(* PLC project static_torsion.project, CODESYS CODESYS V3.5 SP17 Patch 3 *)
(* stored: creationDateTime 1970-01-01T00:00:00, modificationDateTime 2026-06-22T15:12:39.4699931 *)

PROGRAM MODBUS_DATA
  VAR
    MB_DI AT %MW40000 : WORD;  (* Входы дискретные модуль A11 (ECAT-2053) *)
    MB_TN AT %MW40001 : WORD;  (* Значение момента с АЦП модуля тензодатчика A14 (ECAT-2016N) *)
    MB_EN AT %MW40002 : ARRAY[0..1] OF WORD;  (* Угол: измеренное абсолютное значение в условных единицах датчика *)
    MB_DQ AT %MW40004 : WORD;  (* Выходы дискретные модуль A13 (ECAT-2057) (текущее состояние) *)
    MB_STATE AT %MW40005 : WORD;  (* Текущий статус системы управления стендом *)
    MB_TN_OFFSET AT %MW40006 : WORD;  (* Смещение показаний АЦП для коррекции, заданное в ПЛК *)
    MB_EN_OFFSET AT %MW40007 : ARRAY[0..1] OF WORD;  (* Смещение показаний датчика угла, заданное в ПЛК *)
    MB_RD_AUX1 AT %MW40009 : WORD;
    MB_BUF_TN AT %MW40010 : ARRAY[0..(BUFFER_SIZE - 1)] OF WORD;
    MB_HEAD AT %MW40060 : WORD;
    MB_RESERVE AT %MW40061 : ARRAY[0..(BUFFER_SIZE - 1)] OF WORD;
    MB_CTRL AT %MW40111 : WORD;  (* Команда управления режимами работы стенда (основное управление с АРМ) *)
    MB_TORQUE_SV AT %MW40112 : WORD;  (* Задание момента (в масштабированном INT: 25000 = 50 Нм) *)
    MB_VELOCITY_SV AT %MW40113 : WORD;  (* Задание скорости сервопривода (масштабированный INT) *)
    MB_DQ_CTRL AT %MW40114 : WORD;  (* Команда прямого управления дискретными выходами модуль A13 (ECAT-2057) *)
    MB_UZ_CTRL AT %MW40115 : WORD;  (* Команды прямого управления сервоприводом UZ41 *)
    MB_KP AT %MW40116 : ARRAY[0..1] OF WORD;  (* Коэффициенты ПИД регулятора момента: Кп, Ки и Кд соответственно *)
    MB_KI AT %MW40118 : ARRAY[0..1] OF WORD;
    MB_KD AT %MW40120 : ARRAY[0..1] OF WORD;
    MB_TQ_MAX AT %MW40122 : WORD;  (* Аварийная уставка по моменту в Нм (перегорузка при которой привод отключается) *)
    MB_TQ_RANGE AT %MW40123 : WORD;  (* Диапазон датчика момента в Нм (UINT) *)
    MB_ANGLE_SV AT %MW40124 : WORD;  (* Задание угла в градусах *)
    MB_MODEL AT %MW40125 : WORD;  (* Номер модели линеаризации характеристики датчика момента (0 = Линейная модель Y = A * x + B, остальные см. в комментариях) *)
    MB_ANGLE_L AT %MW40126 : WORD;  (* Угол (абсолютный в градусах) ограничения против часовой (крайнее левое положение) *)
    MB_ANGLE_R AT %MW40127 : WORD;  (* Угол (абсолютный в градусах) ограничения по часовой (крайнее правое положение) *)
    MB_A1 AT %MW40128 : ARRAY[0..1] OF WORD;
    MB_B1 AT %MW40130 : ARRAY[0..1] OF WORD;
    MB_C1 AT %MW40132 : ARRAY[0..1] OF WORD;
    MB_A2 AT %MW40134 : ARRAY[0..1] OF WORD;
    MB_B2 AT %MW40136 : ARRAY[0..1] OF WORD;
  END_VAR
  VAR
    _T : WORD_TO_STRUCT;
    _RW : REAL_WORD2;
    ibuff : FB_IntRingBuffer;  (* Кольцевой буфер размером 50 значений для текущих хранения данных от датчика момента *)
    xWriteRetain : R_TRIG;  (* Флаг разрешения записи в энергонезависиимую память *)
  END_VAR
  VAR CONSTANT
    BUFFER_SIZE : UINT := 50;
  END_VAR

            // gen_sin_(PT:=T#1S, AM:=50, OS:= 0, DL:=0);
// Буфер для хранения данных датчика момента
ibuff();
// Обрабатываем данные датчика момента
GVL.rTorque := GetCompensatedTorque(GVL.iTorque_RAW, GVL.iTorque_ADC_offset); // Вычисляем значение датчика момента с учетом начального смещения
GVL.rTorqueCalibrated := GetCalibratedTorque(GVL.rTorque);			// Вычисляем скорректированное значение датчика момента
GVL.iTorqueScaled := CalculateScaledTorque(GVL.rTorqueCalibrated);	// Масштабированное значение для записи в буфер обмена
ibuff.InVal := GVL.iTorqueScaled;									// Добавляем очередное значение в буфер

// ---------- Запись и обработка данных регистров ModbusTCP -------------------
//=============================================================================
// ПЛК -> ПО АРМ
//=============================================================================
MB_DI		 := GVL.DI.WDI;					// Дискретные входы
//-----------------------------------------------------------------------------
MB_TN 		 := TO_WORD(GVL.iTorque_RAW); 	// Данные с АЦП тензодатчика
//-----------------------------------------------------------------------------
MB_EN	 	 := _dint_to_word2(GVL.udiEncoder_RAW); // Энкодер угла
//-----------------------------------------------------------------------------
MB_DQ	 	 := GVL.DQ.WDQ;					// Состояние дискретных выходов
//-----------------------------------------------------------------------------
_T._S_STATE := GVL.State;
MB_STATE    := _T._WORD;		// Статус системы управления
//-----------------------------------------------------------------------------
MB_TN_OFFSET := TO_WORD(GVL.iTorque_ADC_offset); // Смещение 0 АЦП тензодатчика
//-----------------------------------------------------------------------------
MB_EN_OFFSET := _dint_to_word2(GVL.udiEncoderOffset); // Смещение 0 энкодера угла
//-----------------------------------------------------------------------------
MB_BUF_TN 	 := ibuff.Out_WORDS; // Копируем текущие данные буфера датчика в буфер MODBUS
//-----------------------------------------------------------------------------
MB_HEAD 	 := ibuff.head;	 	 // Счетчик позициии указателя на начало текущего буфера

//=============================================================================
// Запись ПО АРМ -> ПЛК
//=============================================================================
IF GVL.fbAlarm.xAlarm THEN
	_T._WORD := MB_CTRL AND 16#FFFE;		// Общая авария, аварийный останов		
ELSE
	_T._WORD := MB_CTRL;		 
END_IF
GVL.Control		:= _T._S_CTRL;	 // Команда управления
//-----------------------------------------------------------------------------
GVL.iTorqueSV	:= TO_INT(MB_TORQUE_SV);		// Задание момента в Нм * 500
//-----------------------------------------------------------------------------
GVL.iJogVelocity := TO_INT(MB_VELOCITY_SV);		// Скорость привода в JOG режиме
												// в град/сек * 1000
//-----------------------------------------------------------------------------
_T._WORD 		:= MB_DQ_CTRL;	 // Прямое управление выходами ПЛК с ПО АРМ
GVL.DQ_Control	:= _T._PDQ;		 // (только в сервисном режиме)
//-----------------------------------------------------------------------------
GVL.UZ_Control 	:=  MB_UZ_CTRL;	// Прямое управление UZ (только в сервисном режиме)

//-----------------------------------------------------------------------------
xWriteRetain(CLK:= GVL.Control.WriteRetain);

IF xWriteRetain.Q THEN
	// Коэффициенты ПИД регулятора
	GVL.KP := _word_to_real(MB_KP);
	GVL.KI := _word_to_real(MB_KI);
	GVL.KD := _word_to_real(MB_KD);
	// Коэффициенты аппроксимации датчика момента
	GVL.rA1 := _word_to_real(MB_A1);
	GVL.rB1 := _word_to_real(MB_B1);
	GVL.rC1 := _word_to_real(MB_C1);
	GVL.rA2 := _word_to_real(MB_A2);
	GVL.rB2 := _word_to_real(MB_B2);
	// Диапазон датчика момента
	GVL.iTorqueSensorRange := 50; //TO_UINT(MB_TQ_RANGE);
END_IF







          
END_PROGRAM
